INTERFACE IExpression EXTENDS __System.IQueryInterface

METHOD IsTrue : BOOL
VAR_INPUT
	i_ptrProcessState: POINTER TO ProcessState;
END_VAR
END_METHOD

METHOD ToString : STRING(256)
VAR_INPUT
END_VAR
END_METHOD

END_INTERFACE

(* stored: Version 1.1.0.1
   Itf IExpression: Id {86b08ee9-b6f2-4b54-aca2-75a34f5eab09}
   Method IsTrue: Id {2b5d3d03-b872-48ba-9bf1-57658319a199}
   Method ToString: Id {c086e87f-8370-4051-9476-f3c5f79dd11d} *)
